ABB RAPID module: Wobj_wobj1_proto1.mod

MODULE Wobj_wobj1_proto1
	! Points are read in order of declaration.
  ! Please do not change the order of points!

  LOCAL PERS robtarget pWobj_U_PointX1:=[[1729.938,-787.0092,168.1094],[0.272077113389969,0.325448632240295,-0.000285798072582111,-0.905570089817047],[-1,-4,2,0],[9E+09,9E+09,9E+09,9E+09,9E+09,9E+09]];
	LOCAL PERS robtarget pWobj_U_PointX2:=[[1743.846,-1396.002,172.9269],[0.272064298391342,0.325436562299728,-0.000269146694336087,-0.905578255653381],[-1,-4,2,0],[9E+09,9E+09,9E+09,9E+09,9E+09,9E+09]];
	LOCAL PERS robtarget pWobj_U_PointY1:=[[1716.74,-781.3937,1144.867],[0.272071003913879,0.325411260128021,-0.00023919006343931,-0.90558534860611],[-1,-4,2,0],[9E+09,9E+09,9E+09,9E+09,9E+09,9E+09]];

ENDMODULE
